PROGRAM z_OVERFLOW

(*-------------------------------------------------------------------------------------------------------*)


(*v025 Ev. Rebosadero*)
MC._07_OVERFLOW.v025_Valv.xOpen:= F_LAVADO_CONT.z_xOverflow;
							
(*V004 Ev. Agua lavado continuo*)
MC._07_OVERFLOW.v004_WaterInlet.xOpen:= F_LAVADO_CONT.z_xLavadoCont;

END_PROGRAM

(* stored: Version 1.1.0.1, ProductVersion 3.1.4024.10
   POU z_OVERFLOW: Id {f62553af-7074-4de8-b8bf-590cad3bfc8f}, SpecialFunc None *)
